Omron CX-Programmer project NewProject (CX-Programmer 9.75)

# PLC ZONE_COMP_PROJECT: CJ2M CPU11

## Global symbols (name address type ; comment)
0.00 BOOL  ; X0
0.01 BOOL  ; S1
0.02 BOOL  ; S2
0.03 BOOL  ; S3
100.00 BOOL  ; FAN 1
100.01 BOOL  ; FAN 2
100.02 BOOL  ; FAN 3

## Program NewProgram1 (cyclic task 0)

### Section Section1

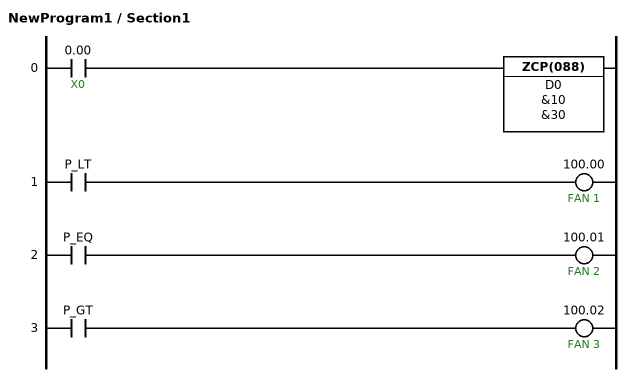
; rung 0
LD 0.00  ; X0
ZCP(088) D0 &10 &30
; rung 1
LD P_LT
OUT 100.00  ; FAN 1
; rung 2
LD P_EQ
OUT 100.01  ; FAN 2
; rung 3
LD P_GT
OUT 100.02  ; FAN 3

### Section END
; rung 0
END(001)